FUNCTION_BLOCK FB_CheckEPS
VAR_IN_OUT
	// Motor that will stop on plc limits
    stMotor	: ST_MotionStage;
	// Array of plc limits and states
    aEPSLimits : ARRAY [*] OF ST_EPSLimits;
END_VAR
VAR_INPUT
	// Encoder Position, Current position of motor. Needed for the case where the motor and encoders are seperate.
	fPosition : REAL;
END_VAR
VAR_OUTPUT
END_VAR
VAR
	nPreviousState : DINT;
	nIndex: DINT;
    nEPSIndex: DINT;
    fbBwdEPS: FB_EPS;
    fbFwdEPS: FB_EPS;
END_VAR

fbBwdEps(eps:=stMotor.stEPSBackwardEnable);
fbFwdEPS(eps:=stMotor.stEPSForwardEnable);

// Look through possible states to see witch state we are in
FOR nIndex := LOWER_BOUND(aEPSLimits, 1) TO UPPER_BOUND(aEPSLimits, 1) BY 1 DO
    IF aEPSLimits[nIndex].stEPS.bEPS_OK THEN
        nEPSIndex := nIndex;
		EXIT; // Stop Looking
    END_IF
END_FOR

IF (NOT (nPreviousState = nEPSIndex)) THEN
	// Clear Previous State Errors
	stMotor.stEPSBackwardEnable.nFlags := 16#FFFFFFFF;
	stMotor.stEPSBackwardEnable.bEPS_OK := TRUE;
	stMotor.stEPSForwardEnable.nFlags := 16#FFFFFFFF;
	stMotor.stEPSForwardEnable.bEPS_OK := TRUE;
END_IF

// Check if position is in plc limit rage
IF fPosition > aEPSLimits[nEPSIndex].fBwd_Limits THEN
	// Winith Limits
    fbBwdEPS.setBit(DINT_TO_BYTE(nEPSIndex), TRUE);
ELSE
	// Outside Limits
    fbBwdEPS.setBit(DINT_TO_BYTE(nEPSIndex), FALSE);
END_IF

IF fPosition < aEPSLimits[nEPSIndex].fFwd_Limits THEN
    fbFwdEPS.setBit(DINT_TO_BYTE(nEPSIndex), TRUE);
ELSE
    fbFwdEPS.setBit(DINT_TO_BYTE(nEPSIndex), FALSE);
END_IF

nPreviousState := nEPSIndex; // Update Previous State

END_FUNCTION_BLOCK

(* stored: Version 1.1.0.1, ProductVersion 3.1.4022.18
   POU FB_CheckEPS: Id {34d78ab9-508b-476a-b7bf-433873b84d5d}, SpecialFunc None *)
